// TIA Portal V19 export
FUNCTION "Pb_Stop_Process" : Void   // FC63, STL
TITLE = Pb - STOP PROCESS (TANK)
{ S7_Optimized_Access := 'TRUE' }
NAME : PBSTTANK
// ****** REVISION HISTORY :
// 
// VERSION DATE         BY    DESCRIPTION
// --------------------------------------------------------------------------
// 00.00   25/9 1997   OPA   ORIGINAL FUNCTION BLOCK
//       
// 00.01    9/2 1998   OPA   START OF "STOP CIP TANK"-PROGRAM ADDED
//                           START OF "TOTAL STOP TANK" IN CIP REMOVED.
//  
// SOFTWARE SIMULATED IN OFFICE *******DATE*********
// stored: AutoNumber false
   VAR_TEMP
      alarmbit : Int;
   END_VAR
BEGIN

NETWORK
TITLE = Pb - STOP PROCESS (TANK)
      A     "LEDAssignment".Stop_AHV_from_scada;  // Stop buttom from scada
      R     "LEDAssignment".Stop_AHV_from_scada;
      JC    M002;

      A     "LEDAssignment".K7_BUTTON;  // "PbK7StopProcess"
      R     "LEDAssignment".K7_BUTTON;  // "PbK7StopProcess"
      JC    M001;
      A     "T 40 RESET STOP LIGHT";
      BEC;
      ON    "LEDAssignment".K7_FLASH;  //"FLASH_K7_STOP"
      O     "LEDAssignment".K7_LIGHT;  //"LIGHT_K7_STOP"
      BEC;
      R     "LEDAssignment".K7_FLASH;  // "FLASH_K7_STOP"
      R     "LEDAssignment".K7_LIGHT;  //"LIGHT_K7_STOP"
      BEU;
M001: AN    "TANK AUTO";
      S     "ProcessAndPbAlarms"."A"[9];  //A09_NoProcessActive// no process active
      L     9;
      JC    Alrm;

//      BEC
      O     "LEDAssignment".K7_FLASH;  //"FLASH_K7_STOP"
      O     "LEDAssignment".K7_LIGHT;  // "LIGHT_K7_STOP"
      JC    M002;
      R     "LEDAssignment".K7_LIGHT;  // "LIGHT_K7_STOP"
      S     "LEDAssignment".K7_FLASH;  // "FLASH_K7_STOP"
      S     "TIM40";
      BEU;
M002: S     "LEDAssignment".K7_FLASH;  // "FLASH_K7_STOP"
      S     "LEDAssignment".K7_LIGHT;  // "LIGHT_K7_STOP"

NETWORK
TITLE = 
      AN    "S0 PRESTERILIZING";
      JC    c001;
      S     "S0 STOP PRESTE. TANK";
      R     "S0 PRESTERILIZING";
      R     "LEDAssignment".K3_FLASH;  //"FLASH_K3_PRESTE."
      R     "LEDAssignment".K3_LIGHT;  //"LIGHT_K3_PRESTE."
      S     "LEDAssignment".K7_FLASH;  //"FLASH_K7_STOP"
      S     "LEDAssignment".K7_LIGHT;  //"LIGHT_K7_STOP"
      BEU;
c001: NOP   0;

NETWORK
TITLE = A10_AllreadyInStopPhase
      AN    "S0 STOP PRESTE. TANK";
      JC    c002;
      S     "ProcessAndPbAlarms"."A"[10];  //A10_AllreadyInStopPhase// already in stop
      L     10;
      JC    Alrm;

//      BEU
c002: NOP   0;

NETWORK
TITLE = A11_TankIsBeingFilled
      AN    "S0 PRODUCTION TANK";
      JC    c003;
      A     "MY0101";
      S     "ProcessAndPbAlarms"."A"[11];  //A11_TankIsBeingFilled// tank is being filled
      L     11;
      R     "LEDAssignment".K7_FLASH;  //"FLASH_K7_STOP"
      R     "LEDAssignment".K7_LIGHT;  //"LIGHT_K7_STOP"
      JC    Alrm;

//      BEC
      S     "S0 STOP PRODUCTION TANK";
      R     "S0 PRODUCTION TANK";
      R     "LEDAssignment".K3_FLASH;  //"FLASH_K3_PRESTE."
      R     "LEDAssignment".K3_LIGHT;  //"LIGHT_K3_PRESTE."
      S     "LEDAssignment".K7_FLASH;  //"FLASH_K7_STOP"
      S     "LEDAssignment".K7_LIGHT;  //"LIGHT_K7_STOP"
      BEU;
c003: NOP   0;

NETWORK
TITLE = A12_NotReadyForTotalStop
      AN    "S0 STOP PRODUCTION TANK";
      JC    c004;
      AN    "LEDAssignment".K4_FLASH;  //"FLASH_K4_CIP_LYE"
      S     "ProcessAndPbAlarms"."A"[12];  //A12_NotReadyForTotalStop// not ready for total stop
      L     12;
      JC    Alrm;

//      BEC
      S     "S0 TOTAL STOP TANK";
      R     "S0 STOP PRODUCTION TANK";
      R     "LEDAssignment".K4_FLASH;  //"FLASH_K4_CIP_LYE"
      R     "LEDAssignment".K4_LIGHT;  //"LIGHT_K4_CIP_LYE"
      R     "LEDAssignment".K5_FLASH;  //"FLASH_K5_CIP_LYE_ACID"
      R     "LEDAssignment".K5_LIGHT;  //"LIGHT_K5_CIP_LYE_ACID"
      BEU;
c004: NOP   0;

NETWORK
TITLE = START: STOP CIP TANK-PROGRAM
// Comment
      AN    "S0 CIP TANK";
      JC    c005;
      S     "S0 STOP CIP TANK";
      R     "S0 CIP TANK";
      R     "LEDAssignment".K4_FLASH;  //"FLASH_K4_CIP_LYE"
      R     "LEDAssignment".K4_LIGHT;  //"LIGHT_K4_CIP_LYE"
      S     "LEDAssignment".K7_FLASH;  //"FLASH_K7_STOP"
      S     "LEDAssignment".K7_LIGHT;  //"LIGHT_K7_STOP"
      R     "LEDAssignment".K5_FLASH;  //"FLASH_K5_CIP_LYE_ACID"
      R     "LEDAssignment".K5_LIGHT;  //"LIGHT_K5_CIP_LYE_ACID"
      BEU;
c005: NOP   0;

NETWORK
TITLE = A10_AllreadyInStopPhase
      AN    "S0 TOTAL STOP TANK";
      JC    c007;
      S     "ProcessAndPbAlarms"."A"[10];  //A10_AllreadyInStopPhase// already in stop
      L     10;
      JC    Alrm;

//      BEC
c007: R     "LEDAssignment".K7_FLASH;  //"FLASH_K7_STOP"
      R     "LEDAssignment".K7_LIGHT;  //"LIGHT_K7_STOP"
      BEU;

NETWORK
TITLE = Blockings alarm text
// Blockings alarm
Alrm: NOP   1;
      T     #alarmbit;
      CALL  "Set_Pop_Up_Blocking"
      ( alarmTextNum := #alarmbit
      );  // start blockings text


END_FUNCTION
